FUNCTION_BLOCK ClearLinkMC EXTENDS FBA_Drive IMPLEMENTS I_EncodedDrive //I_PositionalDrive, I_ContinuousDrive
VAR_OUTPUT
	pulse AT %Q* : INT; //num pulses
	outputRegister AT %Q* : INT;
	brakeRelease AT %Q* : BOOL;
	
	A : BOOL; //direction (F = inwards, T = outwards)
	B : BOOL; //home bit
	clear : BOOL;
	
	hlfb AT %I* : REAL; //high level feedback, if -9999 then servo is idle
	position, targetPos : LREAL;
END_VAR
VAR
	pulseRequest : INT;
	
	minHoming : TON;
	resetTimer : TP;
	
	mode : (DISABLE, HOLD, TARGET, CONTINUOUS, RESET_ERR);
END_VAR
VAR_STAT CONSTANT
	resetTime : TIME := T#1000MS;
	unitsPerPulse : INT := 800; //800 Teknic units per revolution
	distancePerPulse : INT := 5; //5mm per revolution
END_VAR

//M-connector output register
outputRegister.0 := bEnable; 	//enable
outputRegister.1 := A; 			//direction bit
outputRegister.2 := B; 			//homing bit - set to TRUE after startup to begin homing, then set to FALSE to finish homing
outputRegister.3 := clear; 		//reset bit

resetTimer(IN:= , PT:= resetTime, Q=> clear, ET=> ); //reset timer

IF NOT bEnable THEN
	homingComplete := FALSE;
	mode := HOLD;
END_IF

override(); //if sensor limits are reached, this method blocks motion that would exceed the limits

CASE mode OF		
	HOLD: //hold current position, no motion
		pulse := 0;
		pulseRequest := 0;
	
	TARGET:	//target a given position
		IF WithinTolerance(position, targetPos, distancePerPulse) THEN
			pulseRequest := 0;
			mode := HOLD;
			
		ELSIF NOT Busy THEN
			A :=  position < targetPos;
			(*
			2 options to traverse to a target position:
				a)  send all pulses at once - single continuous motion but may exceed limits
				b)  1 pulse at a time - choppy but safer
			*)
			//pulseRequest := TO_INT(ABS(position - targetPos)/distancePerPulse);
			pulseRequest := 1;
			
		END_IF
		
	CONTINUOUS: //single pulses in the direction specified by moveContinuous()
		pulseRequest := 1;
		
	RESET_ERR: //reset pulse, servo may need to be rehomed aftewards
		pulse := 0;
		pulseRequest := 0;
		resetTimer.IN := TRUE;
		
		IF resetTimer.Q THEN
			resetTimer.IN := FALSE;
			mode := HOLD;
		END_IF
		
END_CASE

sequence();

{attribute 'monitoring':='call'}
PROPERTY Busy : BOOL
GET
Busy := hlfb <> -9999;
END_GET
END_PROPERTY

{attribute 'monitoring':='call'}
PROPERTY CurrentPosition : LREAL
GET
CurrentPosition := position;
END_GET
SET
position := CurrentPosition;
END_SET
END_PROPERTY

{attribute 'monitoring':='call'}
PROPERTY Error : BOOL
GET
END_GET
END_PROPERTY

METHOD homingSequence : BOOL
minHoming(IN:= , PT:= T#1S, Q=> , ET=> ); //IN and OUT should be held for at least 1 second - may be removed for deployment

IF NOT bEnable THEN //homing does not begin until software enable
	RETURN;
END_IF

CASE step OF
	Homing.IDLE:
		bEnable := FALSE;
		A := FALSE;
		B := FALSE;
		brakeRelease := TRUE;
		
		homingComplete := FALSE;
		step := Homing.IN;
		
	Homing.IN: //let insertion drop to inner limit before homing
		bEnable := FALSE;
		A := FALSE;
		B := FALSE;
		brakeRelease := TRUE;
		
		minHoming.IN := TRUE;
		
		IF NOT innerLimit AND minHoming.Q THEN
			minHoming.IN := FALSE;
			step := Homing.OUT;
		END_IF
	
	Homing.OUT:
		bEnable := TRUE;
		A := FALSE;
		B := TRUE;
		brakeRelease := TRUE;
		
		minHoming.IN := TRUE;
		
		IF NOT home AND minHoming.Q THEN
			minHoming.IN := FALSE;
			step := Homing.DONE;
		END_IF
		
	Homing.DONE:
		bEnable := TRUE;
		A := FALSE;
		B := FALSE;
		brakeRelease := TRUE;
			
		position := 0;
		
		homingComplete := TRUE;
		homingSequence := TRUE;
		
		mode := HOLD;
		step := Homing.IDLE;
	
END_CASE
END_METHOD

METHOD moveAbsolute : BOOL
VAR_INPUT
	newTarget : LREAL;
END_VAR
targetPos := newTarget;
mode := TARGET;
END_METHOD

METHOD moveContinuous : BOOL
VAR_INPUT
	direction : MC_Direction;
END_VAR
IF direction = MC_Negative_Direction THEN
	A := FALSE;
ELSIF direction = MC_Positive_Direction THEN
	A := TRUE;
END_IF

mode := CONTINUOUS;
END_METHOD

METHOD moveRelative : BOOL
VAR_INPUT
	distance : LREAL;
END_VAR
targetPos := targetPos + distance;

mode := TARGET;
END_METHOD

METHOD PRIVATE override : BOOL
VAR_INPUT
END_VAR
(*
IF (*NOT*) home THEN //block outwards motion
	position := 0;
	IF A THEN
		mode := HOLD;
	END_IF
	
ELSIF (*NOT*) outerLimit AND_THEN A THEN //block outwards motion
	mode := HOLD;

ELSIF (*NOT*) innerLimit AND_THEN NOT A THEN //block inwards motion
	mode := HOLD;
	
END_IF
*)


IF
	((*NOT*) home AND_THEN A) OR
	((*NOT*) outerLimit AND_THEN A) OR
	((*NOT*) innerLimit AND_THEN NOT A)
THEN
	mode := HOLD;
END_IF


IF (*NOT*) home THEN //block outwards motion
	position := 0;
END_IF
END_METHOD

METHOD reset : BOOL
VAR_INPUT
END_VAR
mode := RESET_ERR;
END_METHOD

METHOD PRIVATE sequence : BOOL
VAR_INPUT
END_VAR
IF Busy THEN //servo is active
	IF A THEN //positive direction
		position := position + (distancePerPulse * pulse);
	ELSE //negative direction
		position := position - (distancePerPulse * pulse);
	END_IF
	pulse := 0; //pulses already received, can be set to 0 so position change is not compounded

ELSIF pulse = 0 THEN //servo is not active
	pulse := pulseRequest;
	pulseRequest := 0; //remove this if not working as intended
	
END_IF
END_METHOD

METHOD stop : BOOL
VAR_INPUT
END_VAR
mode := HOLD;
END_METHOD

{attribute 'monitoring':='call'}
PROPERTY TargetPosition : LREAL
GET
END_GET
SET
targetPos := TargetPosition;
END_SET
END_PROPERTY

END_FUNCTION_BLOCK

(* stored: Version 1.1.0.1, ProductVersion 3.1.4024.11
   POU ClearLinkMC: Id {82d395c8-897a-4c3b-989f-b99dc8146760}, SpecialFunc None
   Folder Private: Id {8d4dfb4b-1bc0-44fe-833d-9a6610663d13}
   Folder Properties: Id {f4fb86df-136f-4996-9daa-b3b8a4b4fe75}
   Property Busy: Id {76e617c1-1707-418c-afd8-37e3d0a70099}
   Get Get: Id {9821e814-6021-4995-a4d6-e74adde35b23}
   Property CurrentPosition: Id {552cdbb0-b891-4b67-ad01-a8cfc1c516eb}
   Get Get: Id {f42f05dd-f56e-4930-a286-1888d4d594cd}
   Set Set: Id {cba03562-eb55-4743-94dc-7cf01962b58c}
   Property Error: Id {7daf4b31-4ccd-4ebb-b598-fd16e9795a78}
   Get Get: Id {edbd4fca-a224-4fe5-ba01-ff917580b072}
   Method homingSequence: Id {ed7f9015-f217-4688-b191-db86d43e2b15}
   Method moveAbsolute: Id {dc77def1-bef9-43df-afd0-8ca352bd4ae2}
   Method moveContinuous: Id {56e37924-ed1f-434c-b8b5-86f83bcd5e14}
   Method moveRelative: Id {1770bae9-9ea8-4155-8a6e-b332d1abb598}
   Method override: Id {12f80332-3269-42b5-a267-e03e0f51e546}
   Method reset: Id {b78ab13d-678d-4b52-8830-ac5e90a85d68}
   Method sequence: Id {d3e76146-deb6-4a1c-bf00-057dae828590}
   Method stop: Id {b371037c-73c2-41cf-af60-cf703d5e079a}
   Property TargetPosition: Id {222c0d80-2607-4af6-8461-be098758948d}
   Get Get: Id {b917e1f8-7faf-4ca9-8c30-5bfbcfdfaf97}
   Set Set: Id {f401d7bc-6585-4a9b-ae06-cd3e51203159} *)
